// TwinCAT 3 PLC project PLC1
// Title: Example_project_GSBF
// Company: Gain Automation Technology B.V.
// Author: Gain Automation Technology
// ProjectVersion: 0.0.0.0
// Description: © 2025 Gain Automation Technology B.V. – MIT License
// ProgramVersion: 3.1.4026.19
// libraries:
//   GSBF_Common, * (Gain Automation Technology B.V.)
//   GSBF_HMI, * (Gain Automation Technology B.V.)
//   Tc2_Drive, * (Beckhoff Automation GmbH)
//   Tc2_EtherCAT, * (Beckhoff Automation GmbH)
//   Tc2_MC2, * (Beckhoff Automation GmbH)
//   Tc2_Standard, * (Beckhoff Automation GmbH)
//   Tc2_System, * (Beckhoff Automation GmbH)
//   Tc3_Module, * (Beckhoff Automation GmbH)
//   VisuDialogs, * (System)
//   VisuSymbols, 4.5.0.0 (System)
// project tree:
//   / GlobalTextList.TcGTLO, PlcTask.TcTTO, Visualization Manager.TcVMO (not stored)
//   GVLs/ GVL_Modules.TcGVL
//   POUs/1_Management_Layer/ ST_HmiAlarmList.TcDUT, FB_HMI_AlarmCollector.TcPOU
//   POUs/2_Units/UN_Machine/DUTs/ ST_UN_Machine_Hmi.TcDUT
//   POUs/2_Units/UN_Machine/ UN_Machine.TcPOU
//   POUs/3_Equipment_Modules/EM_InfeedConveyor/ EM_InfeedConveyor.TcPOU
//   POUs/3_Equipment_Modules/EM_InfeedConveyor/_DUTs/ E_EM_InfeedConveyor_Seq_ProductionExecute.TcDUT, E_EM_InfeedConveyor_Seq_ProductionStarting.TcDUT, ST_CommInfeedToLift.TcDUT, ST_CommLiftToInfeed.TcDUT, ST_EM_InfeedConveyor_Hmi.TcDUT
//   POUs/3_Equipment_Modules/EM_Lift/ EM_Lift.TcPOU
//   POUs/3_Equipment_Modules/EM_Lift/_DUTs/ E_EM_Lift_Seq_ProductionExecute.TcDUT, E_EM_Lift_Seq_StopServos.TcDUT, E_EM_Lift_Seq_ProductionStarting.TcDUT, ST_EM_Lift_Hmi.TcDUT
//   POUs/4_Control_Modules/CM_Door/ CM_Door.TcPOU
//   POUs/4_Control_Modules/CM_Door/_DUTs/ E_CM_Door_Seq_Logic.TcDUT, ST_CM_Door_Hmi.TcDUT
//   POUs/6_TwinCatChecks/ CheckBounds.TcPOU, CheckDivDInt.TcPOU, CheckDivLInt.TcPOU, CheckDivLReal.TcPOU, CheckDivReal.TcPOU, CheckLRangeSigned.TcPOU, CheckLRangeUnsigned.TcPOU, CheckPointer.TcPOU, CheckRangeSigned.TcPOU, CheckRangeUnsigned.TcPOU
//   POUs/ MAIN.TcPOU
//   VISUs/ HMI_Button.TcVIS, Header.TcVIS, Page_Main.TcVIS, Page_Alarms.TcVIS, Page_Infeed.TcVIS, Page_PackML.TcVIS, Visualization.TcVIS
// real-time tasks:
//   TASK PlcTask: cycle T#10ms, priority 20, ADS port 350
// motion (NC):
//   TASK NC-Task 1 SAF: cycle T#2ms, priority 4, ADS port 501
//   TASK NC-Task 1 SVB: cycle T#10ms, priority 8, ADS port 511
//   AXIS EM_Lift_Servo (id 1)
//     Dynamic: Jerk=22500
//     OtherSettings: AllowMotionCmdToSlave=true
//     encoder EncType=1
//     drive DrvType=5
//       Analog: TorqueSetpointScale=10, ScaleFactorActTorque=0.1
//       TimeComp: TaskDelayCycles=1
//     controller CtrType=1
//       CtrPara: PriorControlFactor=1
//         Observer: BandWidth=20
//   AXIS EM_LogicExample1_AxisVM (id 2)
//     Dynamic: Jerk=22500
//     OtherSettings: AllowMotionCmdToSlave=true
//     encoder EncType=1
//     drive DrvType=5
//       Analog: TorqueSetpointScale=10, ScaleFactorActTorque=0.1
//       TimeComp: TaskDelayCycles=1
//     controller CtrType=1
//       CtrPara: PriorControlFactor=1
//         Observer: BandWidth=20
//   AXIS EM_LogicExample2_Axis1 (id 4)
//     Dynamic: Jerk=22500
//     OtherSettings: AllowMotionCmdToSlave=true
//     encoder EncType=1
//     drive DrvType=5
//       Analog: TorqueSetpointScale=10, ScaleFactorActTorque=0.1
//       TimeComp: TaskDelayCycles=1
//     controller CtrType=1
//       CtrPara: PriorControlFactor=1
//         Observer: BandWidth=20
//   AXIS EM_LogicExample2_AxisVM (id 3)
//     Dynamic: Jerk=22500
//     OtherSettings: AllowMotionCmdToSlave=true
//     encoder EncType=1
//     drive DrvType=5
//       Analog: TorqueSetpointScale=10, ScaleFactorActTorque=0.1
//       TimeComp: TaskDelayCycles=1
//     controller CtrType=1
//       CtrPara: PriorControlFactor=1
//         Observer: BandWidth=20
// I/O:
//   DEVICE Device 1 (EtherCAT) (disabled), AmsNetId 169.254.247.113.2.1
//     Term 1 (EK1100) [EK1100 EtherCAT Coupler (2A E-Bus)]
//       Term 4 (EL1918) [EL1918, 8Ch. Safety Input 24V, TwinSAFE]
//         modules: Module 2 (FSLOGIC)
//       Term 3 (EL1904) [EL1904, 4 Ch. Safety Input 24V, TwinSAFE]
//         modules: Module 1 (FSOES)
//       Term 2 (EL2912) [EL2912, 2Ch. Safety Output 24V, 2A, TwinSAFE]
//         modules: Module 1 (FSOE), Module 2 (FSOUT), Module 3 (DEVICEIO), Module 4 (FSLOGIC)
// variable links:
//   (this object) <-> Device 1 (EtherCAT)/Term 1 (EK1100)/Term 3 (EL1904)
//     Term 1 (EK1100)/Term 4 (EL1918)/ConnectionInputs/Message_4 TxPDO <-> Module 1 (FSOES)/RxPDO/FSOE
//     Term 1 (EK1100)/Term 4 (EL1918)/ConnectionOutputs/Message_4 RxPDO <-> Module 1 (FSOES)/TxPDO/FSOE
//   (this object) <-> Device 1 (EtherCAT)/Term 1 (EK1100)/Term 4 (EL1918)
//     Term 1 (EK1100)/Term 3 (EL1904)/Module 1 (FSOES)/RxPDO/FSOE <-> ConnectionInputs/Message_4 TxPDO
//     Term 1 (EK1100)/Term 3 (EL1904)/Module 1 (FSOES)/TxPDO/FSOE <-> ConnectionOutputs/Message_4 RxPDO
//   PLC1 Instance <-> NC-Task 1 SAF/Axes/EM_Lift_Servo
//     PlcTask Inputs/GVL_Modules.g_emLift.s_cmMotorLift.IQ_Axis.NcToPlc <-> Outputs/ToPlc
//     PlcTask Outputs/GVL_Modules.g_emLift.s_cmMotorLift.IQ_Axis.PlcToNc <-> Inputs/FromPlc

CONFIGURATION PLC1
    RESOURCE PLC ON TwinCAT3
        TASK PlcTask(INTERVAL := T#10ms, PRIORITY := 20);
        PROGRAM MAIN WITH PlcTask : MAIN;
    END_RESOURCE
END_CONFIGURATION

// ---- POUs/1_Management_Layer/ST_HmiAlarmList.TcDUT
TYPE ST_HmiAlarmList :
STRUCT
	asAlarmList				: ARRAY[1..Param_Alarms.c_nMaxNrOfListEntries] OF STRING; // Active alarm texts for HMI list.
	sHighestActiveAlarm		: STRING; // Highest severity active alarm text.
END_STRUCT
END_TYPE

// ---- POUs/2_Units/UN_Machine/DUTs/ST_UN_Machine_Hmi.TcDUT
TYPE ST_UN_Machine_Hmi :
STRUCT
	// Local var
	fbHmiAlarmCollector		: FB_HMI_AlarmCollector;

END_STRUCT
END_TYPE

// ---- POUs/3_Equipment_Modules/EM_InfeedConveyor/_DUTs/E_EM_InfeedConveyor_Seq_ProductionExecute.TcDUT
{attribute 'qualified_only'}
{attribute 'strict'}
{attribute 'to_string'}
TYPE E_EM_InfeedConveyor_Seq_ProductionExecute :
(
	Idle := c_nSeqIdle, // Wait for production start or preconditions.
	Start := c_nSeqStart, // Select initial step based on sensors/door state.
	
	WaitForProduct, // Wait for product at start sensor.
	
	MoveProductToDoor, // Run belt to move product to end sensor.
	WaitUntilLiftReady, // Wait for lift at infeed position.
	RequestLiftReceiving, // Request lift to receive product.
	OpenDoor, // Open door before transfer.
	MoveProductInLift, // Run belt until lift confirms receipt.
	CloseDoor, // Close door after transfer.
	
	
	
	Ready := c_nSeqReady, // Sequence complete.
	Error := c_nSeqError // Sequence error handling.

);
END_TYPE

// ---- POUs/3_Equipment_Modules/EM_InfeedConveyor/_DUTs/E_EM_InfeedConveyor_Seq_ProductionStarting.TcDUT
{attribute 'qualified_only'}
{attribute 'strict'}
{attribute 'to_string'}
TYPE E_EM_InfeedConveyor_Seq_ProductionStarting :
(
	Idle := c_nSeqIdle, // Wait for PackML start command.
	Start := c_nSeqStart, // Decide open/close door at startup.
	
	OpenDoor, // Open door and wait for feedback.
	CloseDoor, // Close door and wait for feedback.
	
	Ready := c_nSeqReady, // Start sequence complete.
	Error := c_nSeqError // Start sequence error handling.

);
END_TYPE

// ---- POUs/3_Equipment_Modules/EM_InfeedConveyor/_DUTs/ST_CommInfeedToLift.TcDUT
TYPE ST_CommInfeedToLift :
STRUCT
	bReqExportProduct : BOOL; // Request lift to receive product from infeed.
	bBusyWithLift : BOOL; // Infeed busy with lift transfer (handshake/locking).
END_STRUCT
END_TYPE

// ---- POUs/3_Equipment_Modules/EM_InfeedConveyor/_DUTs/ST_CommLiftToInfeed.TcDUT
TYPE ST_CommLiftToInfeed :
STRUCT
	bAtInfeedPos : BOOL; // Lift is positioned at the infeed transfer point.
	bReadyForReceiving : BOOL; // Lift is ready to receive a product.
	bProductReceived : BOOL; // Lift confirms product has been received.
END_STRUCT
END_TYPE

// ---- POUs/3_Equipment_Modules/EM_InfeedConveyor/_DUTs/ST_EM_InfeedConveyor_Hmi.TcDUT
TYPE ST_EM_InfeedConveyor_Hmi :
STRUCT
	fbBelt : HMI_CM_MotorDol; // HMI controls for the infeed belt.
END_STRUCT
END_TYPE

// ---- POUs/3_Equipment_Modules/EM_Lift/_DUTs/E_EM_Lift_Seq_ProductionExecute.TcDUT
{attribute 'qualified_only'}
{attribute 'strict'}
{attribute 'to_string'}
TYPE E_EM_Lift_Seq_ProductionExecute :
(
	Idle := c_nSeqIdle, // Wait for production to start.
	Start := c_nSeqStart, // Begin production sequence steps.

	
	
	Ready := c_nSeqReady, // Sequence complete.
	Error := c_nSeqError // Sequence error handling.

);
END_TYPE

// ---- POUs/3_Equipment_Modules/EM_Lift/_DUTs/E_EM_Lift_Seq_StopServos.TcDUT
{attribute 'qualified_only'}
{attribute 'strict'}
{attribute 'to_string'}
TYPE E_EM_Lift_Seq_StopServos :
(
	Idle := c_nSeqIdle, // Wait for stop request.
	Start := c_nSeqStart, // Begin stop sequence (triggers EMR stop in logic).

	StopServo, // Reserved step for explicit stop if sequence is expanded.
	PowerOffServo, // Remove drive power after stop.
	
	
	Ready := c_nSeqReady, // Stop sequence complete.
	Error := c_nSeqError // Stop sequence error handling.

);
END_TYPE

// ---- POUs/3_Equipment_Modules/EM_Lift/_DUTs/E_EM_Lift_Seq_ProductionStarting.TcDUT
{attribute 'qualified_only'}
{attribute 'strict'}
{attribute 'to_string'}
TYPE E_EM_Lift_Seq_ProductionStarting :
(
	Idle := c_nSeqIdle, // Wait for PackML start command.
	Start := c_nSeqStart, // Decide whether to home or enable drive.
	
	
	ReferenceDrive, // Perform homing/reference procedure.
	EnableDrive, // Power on servo drive.
	MoveToStartPos, // Move to defined start position.
	
	Ready := c_nSeqReady, // Start sequence complete.
	Error := c_nSeqError // Start sequence error handling.

);
END_TYPE

// ---- POUs/3_Equipment_Modules/EM_Lift/_DUTs/ST_EM_Lift_Hmi.TcDUT
TYPE ST_EM_Lift_Hmi :
STRUCT
	fbMotorLift : HMI_CM_Servo; // HMI controls for the lift servo.
END_STRUCT
END_TYPE

// ---- POUs/4_Control_Modules/CM_Door/_DUTs/E_CM_Door_Seq_Logic.TcDUT
{attribute 'qualified_only'}
{attribute 'strict'}
{attribute 'to_string'}
TYPE E_CM_Door_Seq_Logic :
(
	Idle := c_nSeqIdle, // Wait for sequence start.
	Start := c_nSeqStart, // Decide operational vs disabled based on enable.
	
	Disabled, // Module disabled; wait for enable.
	Operational, // Normal door control logic active.
	
	Ready := c_nSeqReady, // Placeholder for ready state (unused in current logic).
	Error := c_nSeqError // Error state; stop motor and wait for clear.
);
END_TYPE

// ---- POUs/4_Control_Modules/CM_Door/_DUTs/ST_CM_Door_Hmi.TcDUT
TYPE ST_CM_Door_Hmi :
STRUCT
	btnCloseDoor : FB_HmiButton; // HMI button: request door close.
	btnOpenDoor : FB_HmiButton; // HMI button: request door open.
	btnStopDoor : FB_HmiButton; // HMI button: request door stop.
	bStaDoorOpen : BOOL; // Status: door open feedback.
	bStaDoorCLosed : BOOL; // Status: door closed feedback.
END_STRUCT
END_TYPE

// ---- GVLs/GVL_Modules.TcGVL
{attribute 'qualified_only'}
VAR_GLOBAL
	
// Management
	g_fbMachCtrlsManager	: FB_MachineControlsManager;
	g_fbHmiMachCtrlsManager	: FB_HMI_MachineControlsManager_StartStopMode;
	g_fbPackMLstatusManager	: FB_PackML_StatusManager;

	
// Units
	g_unMachine				: UN_Machine;
	
// Equipment modules
	g_emInfeedConveyor		: EM_InfeedConveyor;
	g_emLift 				: EM_Lift;
END_VAR

// ---- POUs/MAIN.TcPOU
PROGRAM MAIN 
VAR
END_VAR


// Main program cycle: call top-level managers and units in a clear order.
// Keep this list small; detailed behavior belongs inside the modules.

// PackML status manager
// Collects and aggregates PackML status for the system.
GVL_Modules.g_fbPackMLstatusManager();
	
// Machine controls manager
// HMI manager translates user actions into machine control requests.
GVL_Modules.g_fbHmiMachCtrlsManager(
	i_itfMachineControl := GVL_Modules.g_fbMachCtrlsManager); // Link HMI to machine controls.
// Machine controls manager coordinates PackML state requests for the unit.
GVL_Modules.g_fbMachCtrlsManager(
	i_itfModule := GVL_Modules.g_unMachine); // Link controls to the unit interface.
	
// Units
// Call each unit FB with system-level flags and managers.
GVL_Modules.g_unMachine(
	i_bReqEnable				:= TRUE, // Master enable for the unit (replace with safety chain if needed).
	i_bReqReset					:= GVL_Modules.g_fbMachCtrlsManager.p_bReset, // Reset request from machine controls.
	i_bReqSimulation			:= TRUE, // Simulation mode flag (toggle for real hardware).
	i_itfPackML_Parent			:= GVL_Modules.g_fbPackMLstatusManager, // PackML status manager.
	i_itfAlarmCollector_Parent	:= ); // Optional alarm manager interface.

END_PROGRAM

// ---- POUs/2_Units/UN_Machine/UN_Machine.TcPOU
FUNCTION_BLOCK UN_Machine EXTENDS FB_UN_PackML_Base
VAR_INPUT
END_VAR
VAR_OUTPUT
END_VAR
VAR
	// HMI
	s_stHmi : ST_UN_Machine_Hmi; // HMI structure (status and manual controls).
	
END_VAR

// Call Super
// Basemodule calls the following base method by calling SUPER^(): 
// - m_Main
// Add module-specific cyclic logic before/after SUPER^() if required.

SUPER^();

METHOD PROTECTED _m_Aborted : BOOL (* Return state complete when state is ready*)
VAR_INPUT
	(*First cycle of this state*)
	i_bCmdRestart	: BOOL;
	i_eActMode	: GSBF_Common.E_PackML_Mode;
END_VAR
// Allow clear when alarms are below critical.
// Add extra abort handling here if required.
IF s_fbAlarmCollector.p_eAlarmState < E_Alarm_Severity.Critical THEN
	s_fbPackML.m_ReqClear(); // Request clear of PackML state.
END_IF
END_METHOD

METHOD PROTECTED _m_Alarms
// Call base alarm handling.
SUPER^._m_Alarms();

// Add unit-level alarm conditions here if needed.
END_METHOD

METHOD PROTECTED _m_Hmi
// Call base HMI handling.
SUPER^._m_Hmi();

// Expose alarm collector to HMI for diagnostics.
s_stHmi.fbHmiAlarmCollector(i_itfAlarmCollector := s_fbAlarmCollector);
END_METHOD

METHOD PROTECTED _m_Logic
// Call base logic.
SUPER^._m_Logic();

// Unit-specific logic goes here (coordination between modules).
// Call HMI handling as part of the logic cycle.
_m_Hmi();
END_METHOD

METHOD PROTECTED _m_Modules
// Call base module handling.
SUPER^._m_Modules();

// Call infeed conveyor module and link to lift handshake.
GVL_Modules.g_emInfeedConveyor(
	i_bReqEnable					:= TRUE, // Enable module (replace with safety chain if needed).
	i_bReqReset						:= s_fbAlarmCollector.q_bReqReset, // Reset from alarm collector.
	i_bStaSafetyOk					:= TRUE, // Safety chain OK (replace with real input).
	i_bReqSimulation				:= p_bReqSimulation, // Simulation flag from unit.
	i_itfPackML_Parent				:= s_fbPackML, // PackML parent interface.
	i_itfAlarmCollector_Parent		:= s_fbAlarmCollector, // Alarm collector parent.
	q_stStaPackML					=> , // Optional PackML status feedback.
	i_stFromLift					:= GVL_Modules.g_emLift.q_stFromLift); // Lift status to infeed.

// Call lift module and link to infeed handshake.
GVL_Modules.g_emLift(
	i_bReqEnable:= TRUE, // Enable module (replace with safety chain if needed).
	i_bReqReset:= s_fbAlarmCollector.q_bReqReset, // Reset from alarm collector.
	i_bStaSafetyOk:= TRUE, // Safety chain OK (replace with real input).
	i_bReqSimulation:= p_bReqSimulation, // Simulation flag from unit.
	i_itfPackML_Parent:= s_fbPackML, // PackML parent interface.
	i_itfAlarmCollector_Parent:= s_fbAlarmCollector, // Alarm collector parent.
	q_stStaPackML=> , // Optional PackML status feedback.
	i_stToLift:= GVL_Modules.g_emInfeedConveyor.q_stToLift, // Infeed commands to lift.
	q_stFromLift=> ); // Lift status output.
END_METHOD

METHOD PROTECTED _m_Stopped : BOOL (* Return state complete when state is ready*)
VAR_INPUT
	(*First cycle of this state*)
	i_bCmdRestart	: BOOL;
	i_eActMode	: GSBF_Common.E_PackML_Mode;
END_VAR
// Allow reset when alarms are below error level.
// Add extra stopped-state logic here if required.
IF s_fbAlarmCollector.p_eAlarmState < E_Alarm_Severity.Error THEN
	s_fbPackML.m_ReqReset(); // Request PackML reset.
END_IF
END_METHOD

METHOD PUBLIC m_Main
// Main entry point for the unit.
// Use this to wrap additional high-level logic around base behavior.
SUPER^.m_Main();
END_METHOD

END_FUNCTION_BLOCK

// ---- POUs/3_Equipment_Modules/EM_InfeedConveyor/EM_InfeedConveyor.TcPOU
FUNCTION_BLOCK EM_InfeedConveyor EXTENDS FB_EM_PackML_Base
VAR_INPUT
	i_stFromLift : ST_CommLiftToInfeed; // Status/handshake from lift to infeed.
END_VAR
VAR_OUTPUT
	q_stToLift : ST_CommInfeedToLift; // Commands/handshake from infeed to lift.
END_VAR
VAR
	// Variables
	s_stHmi : ST_EM_InfeedConveyor_Hmi;	// HMI structure (status and manual controls).

	// Control modules
	s_cmBelt : CM_MotorDol; // Belt drive for infeed conveyor.
	s_cmHmiBelt : HMI_CM_MotorDol; // HMI helper for belt controls.
	
	s_cmDoor : CM_Door; // Door control module between conveyor and lift.
	
	
	// in/outputs
	s_diStartConveyor : FB_DigitalInput; // Sensor at conveyor start (product present).
	s_diEndConveyor : FB_DigitalInput; // Sensor at conveyor end (near lift).
	
	// Alarms
	s_fbAlmDoorOpenWithoutPermission : FB_AlarmHandler; // Door open while lift not at infeed.
	s_fbAlmUnexpectProductEndConveyor : FB_AlarmHandler; // Unexpected product detected at end sensor.
	
END_VAR

// Call Super
// Basemodule calls the following base method by calling SUPER^(): 
// - m_Main
// Add module-specific cyclic logic before/after SUPER^() if required.

SUPER^();

METHOD PROTECTED _m_Aborting : BOOL // Return state complete when state is ready
VAR_INPUT
	i_bCmdRestart	: BOOL;	//First cycle of this state
	i_eActMode 		: E_PackML_Mode;
END_VAR
// Stop door.
// Aborting should leave the module in a safe, passive state.
// Add any extra abort actions here (e.g., stop belt, clear outputs).
_m_Aborting	:= s_cmDoor.m_Stop();
END_METHOD

(* Collect alarm conditions from sub-modules. *)
METHOD PROTECTED _m_Alarms
(* All module alarms are handled in this method *)
(*==========================================================================================================*)
// Call base
SUPER^._m_Alarms();

// Add module-specific alarm conditions below.


// Door opened while lift is not at infeed position.
s_fbAlmDoorOpenWithoutPermission(
	i_bCmdRaise:= NOT i_stFromLift.bAtInfeedPos AND NOT s_cmDoor.p_bStaDoorClosed, 
	i_sMessage:= , 
	i_itfAlarmCollector:= p_itfAlarmCollector);

// Unexpected product detected at end sensor (raised explicitly elsewhere).
s_fbAlmUnexpectProductEndConveyor(
	i_bCmdRaise:= , // leave empty, this alarm is set by m_Raise 
	i_sMessage:= , 
	i_itfAlarmCollector:= p_itfAlarmCollector);
END_METHOD

METHOD PROTECTED _m_Execute : BOOL // Return state complete when state is ready
VAR_INPUT
	i_bCmdRestart	: BOOL;	//First cycle of this state
	i_eActMode 		: E_PackML_Mode;
END_VAR
// Execute production sequence only in Production mode.
// For other modes, return TRUE or add mode-specific behavior.
IF i_eActMode = E_PackML_Mode.Production THEN
	_m_Execute := _m_ProductionExecute(i_bCmdRestart := i_bCmdRestart).p_bStaReady;
ELSE
	_m_Execute := TRUE;
END_IF
END_METHOD

METHOD PROTECTED _m_Hmi
// Expose belt controls to the HMI in Manual mode.
// Extend this method with extra HMI controls or status fields as needed.
s_stHmi.fbBelt(
	i_bReqEnableHmiControls:= s_fbPackML.p_eActMode = E_PackML_Mode.Manual, // Enable manual HMI buttons in Manual mode.
	i_itfCM_MotorDol:= s_cmBelt);
END_METHOD

(* Initialization, set initial data. *)
METHOD PROTECTED _m_Init
// Call base
SUPER^._m_Init();

// Configure alarms and initial module parameters here.
// Alarms
s_fbAlmDoorOpenWithoutPermission.p_itfConfig.p_bCfgAutoReset		:= FALSE;                                                
s_fbAlmDoorOpenWithoutPermission.p_itfConfig.p_bCfgEnable			:= TRUE;                                                   
s_fbAlmDoorOpenWithoutPermission.p_itfConfig.p_eCfgSeverity			:= E_Alarm_Severity.Error;                             
s_fbAlmDoorOpenWithoutPermission.p_itfConfig.p_tmCfgDelay			:= T#0S;                                                   
s_fbAlmDoorOpenWithoutPermission.p_itfConfig.p_stCfgEventEntry		:= TC_EVENTs.EM_InfeedConveyor_EventClass.AlmDoorOpenWithoutPermission;

s_fbAlmUnexpectProductEndConveyor.p_itfConfig.p_bCfgAutoReset		:= FALSE;                                                
s_fbAlmUnexpectProductEndConveyor.p_itfConfig.p_bCfgEnable			:= TRUE;                                                   
s_fbAlmUnexpectProductEndConveyor.p_itfConfig.p_eCfgSeverity		:= E_Alarm_Severity.Error;                             
s_fbAlmUnexpectProductEndConveyor.p_itfConfig.p_tmCfgDelay			:= T#0S;                                                   
s_fbAlmUnexpectProductEndConveyor.p_itfConfig.p_stCfgEventEntry		:= TC_EVENTs.EM_InfeedConveyor_EventClass.AlmUnexpectProductEndConveyor;
END_METHOD

(* Process unit inputs. *)
METHOD PROTECTED _m_Inputs
// Call base 
SUPER^._m_Inputs();

// Map IO or communication inputs to internal status here.
// Call inputs
s_diStartConveyor(); // Start sensor at infeed side.
s_diEndConveyor(); // End sensor at lift side.
END_METHOD

(* Call sub-modules (equipment and/or control modules). *)
METHOD PROTECTED _m_Modules
// Call base
SUPER^._m_Modules();

// Call belt motor control module.
s_cmBelt(
	i_bReqEnable:= p_bReqEnable, 
	i_bReqReset:= , // Add extra reset command, normally reset is done by alarmcollector. 
	i_bReqSimulation:= p_bReqSimulation, 
	i_itfAlarmCollector_Parent:= p_itfAlarmCollector); // Propagate belt alarms to module.
	
// Call door control module and pass common flags.
s_cmDoor(
	i_bReqEnable:= p_bReqEnable, 
	i_bReqReset:= , // Add extra reset command, normally reset is done by alarmcollector.
	i_bReqEnableHmiControls:= s_fbPackML.p_eActMode = E_PackML_Mode.Manual, 
	i_bReqSimulation:= p_bReqSimulation, 
	i_itfAlarmCollector_Parent:= p_itfAlarmCollector); // Propagate door alarms to module.
END_METHOD

METHOD _m_ProductionExecute : ITF_FB_SeqControl
VAR_INPUT
	i_bCmdRestart : BOOL;
END_VAR
VAR_INST
	s_fbSeqControl  : FB_SeqControl;
	s_eSeq 			: E_EM_InfeedConveyor_Seq_ProductionExecute;
END_VAR
// Sequencer bookkeeping (current step and entry handling).
s_fbSeqControl(
	i_bReqStart:= i_bCmdRestart, // Start sequencer on first cycle of state.
	i_rnActSeqStep:= s_eSeq, // Active step enum.
	i_sActSeqStep:= TO_STRING(s_eSeq)); // Step name for logging/trace.


// Production sequencer - implement the automatic infeed flow here.
CASE s_eSeq OF
	E_EM_InfeedConveyor_Seq_ProductionExecute.Idle:
		// Wait for production to start or for preconditions.
		// Clear transient outputs here if required (requests, flags).
		;
		
	E_EM_InfeedConveyor_Seq_ProductionExecute.Start:
		// Choose initial step based on current conveyor/door state.
		// This avoids moving product or door unnecessarily at startup.
		IF s_cmDoor.p_bStaDoorClosed AND s_diEndConveyor.p_bStaValue THEN
			// Product already at end and door closed: wait for lift.
			s_fbSeqControl.m_ReqStep(E_EM_InfeedConveyor_Seq_ProductionExecute.WaitUntilLiftReady); // Product at end, wait for lift.
		ELSIF s_cmDoor.p_bStaDoorOpen THEN
			// Door open: request lift to receive immediately.
			s_fbSeqControl.m_ReqStep(E_EM_InfeedConveyor_Seq_ProductionExecute.RequestLiftReceiving);	// Door open, request lift now.
		ELSE
			// Default: wait for product at start sensor.
			s_fbSeqControl.m_ReqStep(E_EM_InfeedConveyor_Seq_ProductionExecute.WaitForProduct);	// Default: wait for product.
		END_IF		
	
	E_EM_InfeedConveyor_Seq_ProductionExecute.WaitForProduct:
		// Wait until a product arrives at the start sensor.
		// Add debouncing or filtering here if required by the hardware.
		IF s_diStartConveyor.p_bStaValue THEN
			s_fbSeqControl.m_ReqStep(E_EM_InfeedConveyor_Seq_ProductionExecute.MoveProductToDoor); // Product detected at start.
		ELSIF s_diEndConveyor.p_bStaValue THEN
			// Product detected at end without running belt -> unexpected.
			s_fbAlmUnexpectProductEndConveyor.m_CmdRaise(); // Raise alarm for unexpected product.
			
			// No transition; PackML will handle the alarm state.
		END_IF
	
	E_EM_InfeedConveyor_Seq_ProductionExecute.MoveProductToDoor:
		// Move product towards the door until end sensor is active.
		// Add jam detection or timeout here if the belt should not run too long.
		IF NOT s_diEndConveyor.p_bStaValue THEN
			// Run belt until product is at end of conveyor.
			s_cmBelt.m_StartFwd(); // Run belt forward.
		ELSE
			// Product is at end conveyor, stop belt.
			IF s_cmBelt.m_Stop() THEN // Stop belt before requesting lift.
				s_fbSeqControl.m_ReqStep(E_EM_InfeedConveyor_Seq_ProductionExecute.WaitUntilLiftReady);
			END_IF
		END_IF
	
	E_EM_InfeedConveyor_Seq_ProductionExecute.WaitUntilLiftReady:
		// Wait until lift is positioned at infeed.
		// Add timeout and alarm handling here if required.
		IF i_stFromLift.bAtInfeedPos THEN
			s_fbSeqControl.m_ReqStep(E_EM_InfeedConveyor_Seq_ProductionExecute.RequestLiftReceiving); // Lift in position.
		END_IF	
			 
	E_EM_InfeedConveyor_Seq_ProductionExecute.RequestLiftReceiving:
		// Handshake: request lift to receive product.
		q_stToLift.bReqExportProduct := TRUE; // Request lift to receive product.
		// Keep this request TRUE while in this step; clear it in other steps if needed.
		
		// Continue once lift confirms it is ready.
		IF i_stFromLift.bReadyForReceiving THEN
			s_fbSeqControl.m_ReqStep(E_EM_InfeedConveyor_Seq_ProductionExecute.OpenDoor); // Lift ready.
		END_IF
		
	E_EM_InfeedConveyor_Seq_ProductionExecute.OpenDoor:
		// Open door before transferring product into lift.
		// Add interlocks here if the door should not open in certain conditions.
		IF s_cmDoor.m_OpenDoor() THEN // Command door open and wait for feedback.
			s_fbSeqControl.m_ReqStep(E_EM_InfeedConveyor_Seq_ProductionExecute.MoveProductInLift);
		END_IF
		
	E_EM_InfeedConveyor_Seq_ProductionExecute.MoveProductInLift:
		// Drive belt until lift reports product received.
		// Add timeout or sensor validation to detect mis-transfer.
		IF NOT i_stFromLift.bProductReceived THEN // Keep feeding until lift confirms receipt.
			// Belt on.
			s_cmBelt.m_StartFwd(); // Move product into lift.
		ELSE	
			// Product in lift, stop conveyor.
			s_cmBelt.m_Stop(); // Stop belt once received.
			
			s_fbSeqControl.m_ReqStep(E_EM_InfeedConveyor_Seq_ProductionExecute.CloseDoor); // Secure door after transfer.
		END_IF
		
	E_EM_InfeedConveyor_Seq_ProductionExecute.CloseDoor:
		// Close door and return to waiting for next product.
		// Add checks for door blocked or safety conditions if required.
		IF s_cmDoor.m_CloseDoor() THEN // Command door close and wait for feedback.
			s_fbSeqControl.m_ReqStep(E_EM_InfeedConveyor_Seq_ProductionExecute.WaitForProduct); // Ready for next product.
		END_IF
		
	E_EM_InfeedConveyor_Seq_ProductionExecute.Ready:
		// Sequence complete; keep outputs stable.
		;
	E_EM_InfeedConveyor_Seq_ProductionExecute.Error:
		// Handle recoverable errors or trigger alarms here.
		;
END_CASE

// Return sequencer status to PackML state handler.
_m_ProductionExecute := s_fbSeqControl.m_getResult(TO_STRING(s_eSeq)); // Return sequencer status.
END_METHOD

METHOD _m_ProductionStarting : ITF_FB_SeqControl
VAR_INPUT
	i_bCmdRestart : BOOL;
END_VAR
VAR_INST
	s_fbSeqControl  : FB_SeqControl;
	s_eSeq 			: E_EM_InfeedConveyor_Seq_ProductionStarting;
END_VAR

// Sequencer bookkeeping (current step and entry handling).
s_fbSeqControl(
	i_bReqStart:= i_bCmdRestart, // Start sequencer on first cycle of state.
	i_rnActSeqStep:= s_eSeq, // Active step enum.
	i_sActSeqStep:= TO_STRING(s_eSeq)); // Step name for logging/trace.
	
// Production start sequence: set door to a known safe state.
CASE s_eSeq OF 
	E_EM_InfeedConveyor_Seq_ProductionStarting.Idle:
		// Wait for start command from PackML.
		// Clear transient outputs here if required (requests, flags).
		;
	E_EM_InfeedConveyor_Seq_ProductionStarting.Start:
		// Decide whether door should be opened or closed at startup.
		// Replace with actual "product present" logic if available.
		IF s_cmDoor.p_bStaDoorBlocked THEN
			s_fbSeqControl.m_ReqStep(E_EM_InfeedConveyor_Seq_ProductionStarting.OpenDoor); // Door blocked, open at start.
		ELSE 
			s_fbSeqControl.m_ReqStep(E_EM_InfeedConveyor_Seq_ProductionStarting.CloseDoor); // Otherwise close at start.
		END_IF
		
		
	E_EM_InfeedConveyor_Seq_ProductionStarting.OpenDoor:
		// Open door at startup (e.g., product present at door).
		// Add interlocks or safety checks here if required.
		IF s_cmDoor.m_OpenDoor() THEN // Command door open and wait for feedback.
			s_fbSeqControl.m_ReqStep(E_EM_InfeedConveyor_Seq_ProductionStarting.Ready); // Startup complete.
		END_IF
	E_EM_InfeedConveyor_Seq_ProductionStarting.CloseDoor:

		// Close door at startup (e.g., no product present).
		// Add interlocks or safety checks here if required.
		IF s_cmDoor.m_CloseDoor() THEN // Command door close and wait for feedback.
			s_fbSeqControl.m_ReqStep(E_EM_InfeedConveyor_Seq_ProductionStarting.Ready); // Startup complete.
		END_IF
		
	E_EM_InfeedConveyor_Seq_ProductionStarting.Ready:
		// Start sequence complete; ready for Execute state.
		;
	E_EM_InfeedConveyor_Seq_ProductionStarting.Error:
		// Handle startup errors or request operator intervention here.
		;
END_CASE

// Return sequencer status to PackML state handler.
_m_ProductionStarting := s_fbSeqControl.m_getResult(TO_STRING(s_eSeq)); // Return sequencer status.
END_METHOD

METHOD PROTECTED _m_Starting : BOOL // Return state complete when state is ready
VAR_INPUT
	i_bCmdRestart	: BOOL;	//First cycle of this state
	i_eActMode 		: E_PackML_Mode;
END_VAR
VAR_INST
	s_fbSeqControl 	: FB_SeqControl;
	s_eSeq			: E_EM_InfeedConveyor_Seq_ProductionStarting;
END_VAR
// PackML Starting: run production-start sequencer in Production mode.
IF i_eActMode = E_PackML_Mode.Production THEN
	_m_Starting := _m_ProductionStarting(i_bCmdRestart := i_bCmdRestart).p_bStaReady;
ELSE
	_m_Starting := TRUE;
END_IF
END_METHOD

METHOD PROTECTED _m_Stopping : BOOL // Return state complete when state is ready
VAR_INPUT
	i_bCmdRestart	: BOOL;	//First cycle of this state
	i_eActMode 		: E_PackML_Mode;
END_VAR
// Stop door.
// Add belt stop or other safe-state actions if required.
_m_Stopping	:= s_cmDoor.m_Stop();
END_METHOD

END_FUNCTION_BLOCK

// ---- POUs/4_Control_Modules/CM_Door/CM_Door.TcPOU
FUNCTION_BLOCK CM_Door EXTENDS FB_CM_Base
VAR_INPUT
	i_bReqEnableHmiControls : BOOL;	// Request to enable HMI control buttons (open/close/stop).
END_VAR
VAR_OUTPUT
END_VAR
VAR
	// Control modules
	s_cmMotor : CM_MotorDol; // Door motor (forward=open, reverse=close).
 
	
	// in/outputs
	s_diDoorIsOpen : FB_DigitalInput; // Feedback: door open position.
	s_diDoorIsClosed : FB_DigitalInput; // Feedback: door closed position.
	s_diDoorIsBlocked : FB_DigitalInput; // Feedback: door blocked sensor.
	
	// Alarms
	
	s_fbAlmDoorIsBlocked : FB_AlarmHandler; // Blocked while moving.
	s_fbAlmFeedbackBothOn : FB_AlarmHandler; // Both open and closed feedback active.
	s_fbAlmDoorNotOpen : FB_AlarmHandler; // Door did not reach open position.
	s_fbAlmDoorNotClosed : FB_AlarmHandler;	// Door did not reach closed position.

	// Hmi
	s_stHmi : ST_CM_Door_Hmi; // HMI structure (buttons + status).
END_VAR

// Call base 
SUPER^();

(* Monitor alarm conditions. *)
METHOD PROTECTED _m_Alarms

SUPER^._m_Alarms();

// Feedback conflict: open and closed at the same time.
s_fbAlmFeedbackBothOn(
	i_bCmdRaise:= s_diDoorIsOpen.p_bStaValue AND s_diDoorIsClosed.p_bStaValue, 
	i_sMessage:= , 
	i_itfAlarmCollector:= p_itfAlarmCollector);
	
// Door blocked while motor runs.
s_fbAlmDoorIsBlocked(
	i_bCmdRaise:= NOT s_cmMotor.p_bStaStandstill AND s_diDoorIsBlocked.p_bStaValue, 
	i_sMessage:= , 
	i_itfAlarmCollector:= p_itfAlarmCollector);
	
// Door should open within delay when running forward.
s_fbAlmDoorNotOpen.p_itfConfig.p_tmCfgDelay := T#6S;	
s_fbAlmDoorNotOpen(
	i_bCmdRaise:= s_cmMotor.p_bStaRunningFwd AND NOT s_diDoorIsOpen.p_bStaValue, 
	i_sMessage:= , 
	i_itfAlarmCollector:= p_itfAlarmCollector);
	

// Door should close within delay when running reverse.
s_fbAlmDoorNotClosed.p_itfConfig.p_tmCfgDelay := T#6S;		
s_fbAlmDoorNotClosed(
	i_bCmdRaise:= s_cmMotor.p_bStaRunningRev AND NOT s_diDoorIsClosed.p_bStaValue, 
	i_sMessage:= , 
	i_itfAlarmCollector:= p_itfAlarmCollector);
END_METHOD

METHOD PROTECTED _m_Hmi
VAR_INPUT
END_VAR
VAR_INST
	s_bStaOpening : BOOL;
	s_bStaClosing : BOOL;
END_VAR



// Update HMI buttons with current enable/state.
s_stHmi.btnOpenDoor(
	i_bEnable:= i_bReqEnableHmiControls, 
	i_bProcessState:= s_bStaOpening);
	
s_stHmi.btnCloseDoor(
	i_bEnable:= i_bReqEnableHmiControls, 
	i_bProcessState:= s_bStaClosing);

s_stHmi.btnStopDoor(
	i_bEnable:= i_bReqEnableHmiControls);	
	
// Latch requested direction on rising edge.
IF s_stHmi.btnOpenDoor.q_bStateOsr THEN
	s_bStaOpening := TRUE;
	s_bStaClosing := FALSE;
END_IF	

IF s_stHmi.btnCloseDoor.q_bStateOsr THEN
	s_bStaOpening := FALSE;
	s_bStaClosing := TRUE;
END_IF	

// Stop request or error cancels movement.
IF s_stHmi.btnStopDoor.q_bStateOsr OR p_eAlarmState >= E_Alarm_Severity.Error THEN
	s_bStaOpening := FALSE;
	s_bStaClosing := FALSE;
	m_Stop();
END_IF	

// Execute open/close request until feedback is reached.
IF s_bStaOpening THEN
	IF m_OpenDoor() THEN
		s_bStaOpening := FALSE;
	END_IF
END_IF


IF s_bStaClosing THEN
	IF m_CloseDoor() THEN
		s_bStaClosing := FALSE;
	END_IF
END_IF

// Publish status to HMI.
s_stHmi.bStaDoorOpen := p_bStaDoorOpen;
s_stHmi.bStaDoorCLosed := p_bStaDoorClosed;
END_METHOD

(* Initialization, set initial data. *)
METHOD PROTECTED _m_Init
// Call base
SUPER^._m_Init();

// Alarms
s_fbAlmDoorIsBlocked.p_itfConfig.p_bCfgAutoReset		:= FALSE;                                                
s_fbAlmDoorIsBlocked.p_itfConfig.p_bCfgEnable			:= TRUE;                                                   
s_fbAlmDoorIsBlocked.p_itfConfig.p_eCfgSeverity			:= E_Alarm_Severity.Error;                             
s_fbAlmDoorIsBlocked.p_itfConfig.p_tmCfgDelay			:= T#0S;                                                   
s_fbAlmDoorIsBlocked.p_itfConfig.p_stCfgEventEntry		:= TC_EVENTS.Alarmen.CM_Door_AlmDoorIsBlocked;

s_fbAlmFeedbackBothOn.p_itfConfig.p_bCfgAutoReset		:= FALSE;                                                
s_fbAlmFeedbackBothOn.p_itfConfig.p_bCfgEnable			:= TRUE;                                                   
s_fbAlmFeedbackBothOn.p_itfConfig.p_eCfgSeverity			:= E_Alarm_Severity.Error;                             
s_fbAlmFeedbackBothOn.p_itfConfig.p_tmCfgDelay			:= T#0S;                                                   
s_fbAlmFeedbackBothOn.p_itfConfig.p_stCfgEventEntry		:= TC_EVENTS.Alarmen.CM_Door_AlmFeedbackBothOn;

s_fbAlmDoorNotOpen.p_itfConfig.p_bCfgAutoReset			:= FALSE;                                                
s_fbAlmDoorNotOpen.p_itfConfig.p_bCfgEnable				:= TRUE;                                                   
s_fbAlmDoorNotOpen.p_itfConfig.p_eCfgSeverity			:= E_Alarm_Severity.Error;                             
s_fbAlmDoorNotOpen.p_itfConfig.p_tmCfgDelay				:= T#0S;                                                   
s_fbAlmDoorNotOpen.p_itfConfig.p_stCfgEventEntry		:= TC_EVENTs.Alarmen.CM_Door_AlmDoorIsBlocked;

s_fbAlmDoorNotClosed.p_itfConfig.p_bCfgAutoReset		:= FALSE;                                                
s_fbAlmDoorNotClosed.p_itfConfig.p_bCfgEnable			:= TRUE;                                                   
s_fbAlmDoorNotClosed.p_itfConfig.p_eCfgSeverity			:= E_Alarm_Severity.Error;                             
s_fbAlmDoorNotClosed.p_itfConfig.p_tmCfgDelay			:= T#0S;                                                   
s_fbAlmDoorNotClosed.p_itfConfig.p_stCfgEventEntry		:= TC_EVENTs.Alarmen.CM_Door_AlmFeedbackBothOn;
END_METHOD

(* Read hardware and module inputs. If applicable, apply filtering, scaling and/or conversion to local variables. *) 
METHOD PROTECTED _m_Inputs
// Call base
SUPER^._m_Inputs();


// Call inputs
s_diDoorIsOpen();
s_diDoorIsClosed();
s_diDoorIsBlocked();
END_METHOD

(* Handle the internal logic of the control module. *)
METHOD PROTECTED _m_Logic
VAR_INST
	s_fbSeqControl : FB_SeqControl;
	s_eSeq : E_CM_Door_Seq_Logic;
END_VAR
// Call base
SUPER^._m_Logic();

_m_Hmi();

// Call modules
_m_Modules();

// Sequencer tracks the door state machine.
// Call sequencer
s_fbSeqControl(
	i_bReqStart:= FALSE, 
	i_rnActSeqStep:= s_eSeq, 
	i_sActSeqStep:= TO_STRING(s_eSeq));

// Logic
CASE s_eSeq OF 
	E_CM_Door_Seq_Logic.Idle:
		// Go to operational state
		s_fbSeqControl.m_ReqStep(E_CM_Door_Seq_Logic.Start);
		
	E_CM_Door_Seq_Logic.Start:

		IF NOT p_bReqEnable THEN
			// Disabled request takes priority.
			s_fbSeqControl.m_ReqStep(E_CM_Door_Seq_Logic.Disabled);
		ELSE
			// Start successful: go operational.
			s_fbSeqControl.m_ReqStep(E_CM_Door_Seq_Logic.Operational);
		END_IF
	
	E_CM_Door_Seq_Logic.Disabled:
		IF p_bReqEnable THEN
			// Re-enable sequence.
			s_fbSeqControl.m_ReqStep(E_CM_Door_Seq_Logic.Start);
		END_IF
	
		
	E_CM_Door_Seq_Logic.Operational:
		// Stop motor when door is open
		IF s_diDoorIsOpen.p_bStaValue 
			AND s_cmMotor.p_bStaRunningFwd 
		THEN
			m_Stop();
		END_IF
		
		// Stop motor when door is closed
		IF s_diDoorIsClosed.p_bStaValue 
			AND s_cmMotor.p_bStaRunningRev 
		THEN
			m_Stop();
		END_IF
		
	
	
		// Transition
		IF NOT p_bReqEnable THEN
			// Disabled request wins.
			s_fbSeqControl.m_ReqStep(E_CM_Door_Seq_Logic.Disabled);
		ELSIF p_eAlarmState >= E_Alarm_Severity.Error THEN
			// Some error is active, go to error state
			s_fbSeqControl.m_ReqStep(E_CM_Door_Seq_Logic.Error);
		END_IF


	
	E_CM_Door_Seq_Logic.Ready:
		;
		
	E_CM_Door_Seq_Logic.Error:
		// Stop motor
		m_Stop();
	
		// Transition 
		IF NOT p_bReqEnable THEN
			s_fbSeqControl.m_ReqStep(E_CM_Door_Seq_Logic.Disabled);
		ELSIF p_eAlarmState < E_Alarm_Severity.Error THEN
			// Error cleared: restart sequence.
			s_fbSeqControl.m_ReqStep(E_CM_Door_Seq_Logic.Start);
		END_IF

END_CASE

s_fbSeqControl.m_Update(i_sActSeqStep := TO_STRING(s_eSeq));
END_METHOD

METHOD _m_Modules : BOOL
VAR_INPUT
END_VAR
// Call motor control module and connect to alarm collector.
s_cmMotor(
	i_bReqEnable:= p_bReqEnable, 
	i_bReqReset:= , // Can be leaved empty, is automatically done by alarmcollector
	i_bReqSimulation:= i_bReqSimulation, 
	i_itfAlarmCollector_Parent:= p_itfAlarmCollector);
END_METHOD

METHOD PROTECTED _m_Simulation
VAR_INST
	s_bSimDoorIsClosed : BOOL;
	s_bSimDoorIsOpen : BOOL;
	
	s_tonSimOpening : TON;
	s_tonSimClosing : TON;
END_VAR


// Simulate feedback timing based on motor direction.
s_tonSimOpening(in := s_cmMotor.p_bStaRunningFwd, PT := T#1MS);
s_tonSimClosing(in := s_cmMotor.p_bStaRunningRev, PT := T#5MS);

// When motor is running for x seconds set simulation status to open. 
IF s_tonSimOpening.Q THEN
	s_bSimDoorIsOpen := TRUE;
ELSIF s_cmMotor.p_bStaRunningRev THEN
	s_bSimDoorIsOpen := FALSE;	
END_IF

// When motor is running reverse long enough set simulation status to closed.
IF s_tonSimClosing.Q THEN
	s_bSimDoorIsClosed := TRUE;
ELSIF s_cmMotor.p_bStaRunningFwd THEN
	s_bSimDoorIsClosed := FALSE;	
END_IF

// Copy simulation value to IO
s_diDoorIsOpen.m_Simulation(i_bSimulate := p_bReqSimulation, i_bvalue := s_bSimDoorIsOpen);
s_diDoorIsClosed.m_Simulation(i_bSimulate := p_bReqSimulation, i_bvalue := s_bSimDoorIsClosed);
END_METHOD

METHOD m_CloseDoor : BOOL
VAR_INPUT
END_VAR
// Run reverse until closed feedback is active.
IF p_bReqEnable 
	AND p_eAlarmState < E_Alarm_Severity.Error 
	AND NOT s_diDoorIsClosed.p_bStaValue 
THEN
	// Start motor reverse
	s_cmMotor.m_StartRev();
ELSE
	s_cmMotor.m_Stop();
END_IF

m_CloseDoor := s_diDoorIsClosed.p_bStaValue;
END_METHOD

METHOD m_OpenDoor : BOOL
VAR_INPUT
END_VAR
// Run forward until open feedback is active.
IF p_bReqEnable 
	AND p_eAlarmState < E_Alarm_Severity.Error 
	AND NOT s_diDoorIsOpen.p_bStaValue 
THEN
	// Start motor forward
	s_cmMotor.m_StartFwd();
ELSE
	s_cmMotor.m_Stop();
END_IF

m_OpenDoor := s_diDoorIsOpen.p_bStaValue;
END_METHOD

METHOD m_Stop : BOOL
VAR_INPUT
END_VAR
// Stop motor and report standstill.
s_cmMotor.m_Stop();

m_Stop := s_cmMotor.p_bStaStandstill;
END_METHOD

PROPERTY p_bStaDoorBlocked : BOOL
GET
p_bStaDoorBlocked := s_diDoorIsBlocked.p_bStaValue;
END_GET
END_PROPERTY

PROPERTY PUBLIC p_bStaDoorClosed : BOOL
GET
p_bStaDoorClosed := s_diDoorIsClosed.p_bStaValue;
END_GET
END_PROPERTY

PROPERTY PUBLIC p_bStaDoorOpen : BOOL
GET
p_bStaDoorOpen := s_diDoorIsOpen.p_bStaValue;
END_GET
END_PROPERTY

END_FUNCTION_BLOCK

// ---- POUs/3_Equipment_Modules/EM_Lift/EM_Lift.TcPOU
FUNCTION_BLOCK EM_Lift EXTENDS FB_EM_PackML_Base
VAR_INPUT
	i_stToLift : ST_CommInfeedToLift; // Command from infeed to lift.
END_VAR
VAR_OUTPUT
	q_stFromLift : ST_CommLiftToInfeed; // Status from lift to infeed.
END_VAR
VAR
	// Variables
	s_stHmi : ST_EM_Lift_Hmi;	// HMI status and controls.


	// Control modules
	s_cmMotorLift : CM_ServoAX8000;	// Lift servo axis control.
	
END_VAR

// Call Super
// Basemodule calls the following base method by calling SUPER^(): 
// - m_Main
// Add module-specific cyclic logic before/after SUPER^() if required.

SUPER^();

METHOD PROTECTED _m_Aborting : BOOL // Return state complete when state is ready
VAR_INPUT
	i_bCmdRestart	: BOOL;	//First cycle of this state
	i_eActMode 		: E_PackML_Mode;
END_VAR
// Abort and disable servo
// Use stop-sequence to bring the lift axis to a safe state.
// Add any extra abort actions here (e.g., vent valves, set outputs).
_m_Aborting	:= _m_SeqStopServos(i_bCmdRestart := i_bCmdRestart).p_bStaReady;
END_METHOD

(* Collect alarm conditions from sub-modules. *)
METHOD PROTECTED _m_Alarms
(* All module alarms are handled in this method *)
(*==========================================================================================================*)
// Call base
SUPER^._m_Alarms();

// Add module-specific alarm conditions here and link them to the alarm collector.
END_METHOD

METHOD PROTECTED _m_Execute : BOOL // Return state complete when state is ready
VAR_INPUT
	i_bCmdRestart	: BOOL;	//First cycle of this state
	i_eActMode 		: E_PackML_Mode;
END_VAR
// Execute production sequence only in Production mode.
// For other modes, return TRUE or add mode-specific logic.
IF i_eActMode = E_PackML_Mode.Production THEN
	_m_Execute := _m_ProductionExecute(i_bCmdRestart := i_bCmdRestart).p_bStaReady;
ELSE
	_m_Execute := TRUE;
END_IF
END_METHOD

METHOD PROTECTED _m_Hmi
// Expose lift servo controls to the HMI in Manual mode.
// Extend this method with extra HMI widgets or status fields as needed.
s_stHmi.fbMotorLift(
	i_bReqEnableHmiControls:= s_fbPackML.p_eActMode = E_PackML_Mode.Manual, 
	i_itfCM_Servo:= s_cmMotorLift,
	i_eCfgMoveAbs:= E_HMI_CM_SERVO_MoveAbsMode_Direction.MoveToModuloPosShortestWay);
END_METHOD

(* Initialization, set initial data. *)
METHOD PROTECTED _m_Init
// Call base
SUPER^._m_Init();

// Initialize module-specific parameters and defaults here.
END_METHOD

(* Process unit inputs. *)
METHOD PROTECTED _m_Inputs
// Call base 
SUPER^._m_Inputs();

// Map IO or communication inputs to internal variables here.
END_METHOD

(* Call sub-modules (equipment and/or control modules). *)
METHOD PROTECTED _m_Modules
// Call base
SUPER^._m_Modules();

// Call lift servo control module and pass common flags.
// Adjust override, interlocks, and safety conditions to your machine.
s_cmMotorLift(
	i_bReqEnable:= p_bReqEnable, // Enable/reset/simulation are typically controlled by PackML/base module.
	i_bReqReset:= ,				 // done by alarmcollector 
	i_bReqSimulation:= p_bReqSimulation, 	// Connect alarm collector so servo alarms propagate to the module.
	i_itfAlarmCollector_Parent:= s_fbAlarmCollector, 
	i_bEmrStopOk:= TRUE, // Safety chain OK (replace with real E-Stop OK signal if available)
	i_fOverride:= 100, // Motion override in percent (100 = full speed).
	i_bDisableForward:= FALSE, // Direction/axis interlocks (set TRUE to block motion).
	i_bDisableReverse:= FALSE, // Direction/axis interlocks (set TRUE to block motion).
	i_bDisableAxis:= FALSE, 
	i_bExtReferenceSignal:= );	// Optional external reference signal (leave empty if unused).
END_METHOD

METHOD _m_ProductionExecute : ITF_FB_SeqControl
VAR_INPUT
	i_bCmdRestart : BOOL;
END_VAR
VAR_INST
	s_fbSeqControl  : FB_SeqControl;
	s_eSeq 			: E_EM_Lift_Seq_ProductionExecute;
END_VAR
// Sequencer bookkeeping (current step and entry handling).
s_fbSeqControl(
	i_bReqStart:= i_bCmdRestart, 
	i_rnActSeqStep:= s_eSeq, 
	i_sActSeqStep:= TO_STRING(s_eSeq));


// Production sequencer - implement the automatic process here.
CASE s_eSeq OF
	E_EM_Lift_Seq_ProductionExecute.Idle:
		// Wait for start conditions or upstream handshake.
		;
		
	E_EM_Lift_Seq_ProductionExecute.Start:
		// Add first motion/command steps for the production cycle.
		;
		
	E_EM_Lift_Seq_ProductionExecute.Ready:
		// Sequence complete; state complete is set automatically to omac.
		;
	E_EM_Lift_Seq_ProductionExecute.Error:
		;
END_CASE

// Return sequencer status to PackML state handler.
_m_ProductionExecute := s_fbSeqControl.m_getResult(TO_STRING(s_eSeq));
END_METHOD

METHOD _m_ProductionStarting : ITF_FB_SeqControl
VAR_INPUT
	i_bCmdRestart : BOOL;
END_VAR
VAR_INST
	s_fbSeqControl  : FB_SeqControl;
	s_eSeq 			: E_EM_Lift_Seq_ProductionStarting;
	s_stHomingOptions : ST_HomingOptions;
END_VAR

// Sequencer bookkeeping (current step and entry handling).
s_fbSeqControl(
	i_bReqStart:= i_bCmdRestart, 
	i_rnActSeqStep:= s_eSeq, 
	i_sActSeqStep:= TO_STRING(s_eSeq));
	
// Production start sequence: home, enable, and move to a known start position.
CASE s_eSeq OF 
	E_EM_Lift_Seq_ProductionStarting.Idle:
		// Wait for start command from PackML.
		;
	E_EM_Lift_Seq_ProductionStarting.Start:
		// Current logic: if axis reports homed, re-run reference; otherwise enable.
		// Adjust this decision to match your homing policy.
		IF s_cmMotorLift.p_bStaHomed THEN
			s_fbSeqControl.m_ReqStep(E_EM_Lift_Seq_ProductionStarting.ReferenceDrive);
		ELSE	
			s_fbSeqControl.m_ReqStep(E_EM_Lift_Seq_ProductionStarting.EnableDrive);
		END_IF
	
	E_EM_Lift_Seq_ProductionStarting.ReferenceDrive:
		// Configure homing behavior for this axis.
		s_stHomingOptions.ClearPositionLag := TRUE;
		s_stHomingOptions.SearchDirection := MC_Direction.MC_Positive_Direction;
		s_stHomingOptions.SearchVelocity := 500;
		s_stHomingOptions.SyncDirection := MC_Direction.MC_Negative_Direction;
		s_stHomingOptions.SyncVelocity := 100;
		s_stHomingOptions.ReferenceMode := E_EncoderReferenceMode.ENCODERREFERENCEMODE_DEFAULT;
		
		// Start homing on entry and wait until it completes.
		IF s_cmMotorLift.m_Home(
			i_bCmdExecute:= s_fbSeqControl.p_bStaEntry, 
			i_bForceReference:= TRUE, 
			i_eHomingMode:= MC_HomingMode.MC_Direct, 
			i_eBufferMode:= MC_BufferMode.MC_Aborting, 
			i_fPosition:= 0.0, 
			i_stOptions:= s_stHomingOptions, 
			i_sLogHint:= 'Starting')
		THEN
			s_fbSeqControl.m_ReqStep(E_EM_Lift_Seq_ProductionStarting.EnableDrive);
		END_IF
	E_EM_Lift_Seq_ProductionStarting.EnableDrive:
		// Power on the drive before any absolute move commands.
		IF s_cmMotorLift.m_PowerOn() THEN
			s_fbSeqControl.m_ReqStep(E_EM_Lift_Seq_ProductionStarting.MoveToStartPos);
		END_IF
		
	E_EM_Lift_Seq_ProductionStarting.MoveToStartPos:
		// Move to a defined start position for production.
		IF s_cmMotorLift.m_MoveAbsolute(
								i_bCmdExecute:= s_fbSeqControl.p_bStaEntry, 
								i_fAcceleration:= 500, 
								i_fDeceleration:= 500, 
								i_fJerk:= 5000, 
								i_fSpeed:= 100, 
								i_fPosition:= 100, 
								i_eBufferMode:= MC_BufferMode.MC_Aborting, 
								i_sLogHint:= 'Starting, move to startposition')	
		THEN
			s_fbSeqControl.m_ReqStep(E_EM_Lift_Seq_ProductionStarting.Ready);
		END_IF
		
	E_EM_Lift_Seq_ProductionStarting.Ready:
		// Start sequence complete; ready for Execute state.
		;
	E_EM_Lift_Seq_ProductionStarting.Error:
		;
END_CASE

// Return sequencer status to PackML state handler.
_m_ProductionStarting := s_fbSeqControl.m_getResult(TO_STRING(s_eSeq));
END_METHOD

METHOD _m_SeqStopServos : ITF_FB_SeqControl
VAR_INPUT
	i_bCmdRestart : BOOL;
END_VAR
VAR_INST
	s_fbSeqControl  : FB_SeqControl;
	s_eSeq 			: E_EM_Lift_Seq_StopServos;
END_VAR
// Sequencer bookkeeping (current step and entry handling).
s_fbSeqControl(
	i_bReqStart:= i_bCmdRestart, 
	i_rnActSeqStep:= s_eSeq, 
	i_sActSeqStep:= TO_STRING(s_eSeq));


// Stop sequence - bring the servo to a safe, powered-off state.
CASE s_eSeq OF
	E_EM_Lift_Seq_StopServos.Idle:
		// Wait for stop request from PackML or safety logic.
		;
		
	E_EM_Lift_Seq_StopServos.Start:
		// Issue emergency stop to decelerate as fast as possible.
		IF s_cmMotorLift.m_EmrStop(i_bCmdExecute := s_fbSeqControl.p_bStaEntry) THEN
			s_fbSeqControl.m_ReqStep(E_EM_Lift_Seq_StopServos.PowerOffServo);
		ELSIF s_fbSeqControl.p_tmStepTime > T#200MS THEN	
			// Not stopped in expected time; continue with power-off.
			s_fbSeqControl.m_ReqStep(E_EM_Lift_Seq_StopServos.PowerOffServo);
		END_IF
		
	E_EM_Lift_Seq_StopServos.PowerOffServo :	
		// Remove drive power after the stop request.
		IF s_cmMotorLift.m_PowerOff() THEN
			s_fbSeqControl.m_ReqStep(E_EM_Lift_Seq_StopServos.Ready);
		ELSIF s_fbSeqControl.p_tmStepTime > T#200MS THEN
			// Not powered off in expected time; end sequence anyway.
			s_fbSeqControl.m_ReqStep(E_EM_Lift_Seq_StopServos.Ready);
		END_IF
			
		
	E_EM_Lift_Seq_StopServos.Ready:
		// Stop sequence complete.
		;
	E_EM_Lift_Seq_StopServos.Error:
		;
END_CASE

// Return sequencer status to PackML state handler.
_m_SeqStopServos := s_fbSeqControl.m_getResult(TO_STRING(s_eSeq));
END_METHOD

METHOD PROTECTED _m_Starting : BOOL // Return state complete when state is ready
VAR_INPUT
	i_bCmdRestart	: BOOL;	//First cycle of this state
	i_eActMode 		: E_PackML_Mode;
END_VAR
VAR_INST
	s_fbSeqControl 	: FB_SeqControl;
	s_eSeq			: E_EM_InfeedConveyor_Seq_ProductionStarting;
END_VAR
// PackML Starting: run production-start sequencer in Production mode.
IF i_eActMode = E_PackML_Mode.Production THEN
	_m_Starting := _m_ProductionStarting(i_bCmdRestart := i_bCmdRestart).p_bStaReady;
ELSE
	_m_Starting := TRUE;
END_IF
END_METHOD

METHOD PROTECTED _m_Stopping : BOOL // Return state complete when state is ready
VAR_INPUT
	i_bCmdRestart	: BOOL;	//First cycle of this state
	i_eActMode 		: E_PackML_Mode;
END_VAR
// Abort and disable servo
// PackML Stopping reuses the stop-sequence to safely disable the servo.
_m_Stopping	:= _m_SeqStopServos(i_bCmdRestart := i_bCmdRestart).p_bStaReady;
END_METHOD

END_FUNCTION_BLOCK

// ---- POUs/1_Management_Layer/FB_HMI_AlarmCollector.TcPOU
FUNCTION_BLOCK FB_HMI_AlarmCollector EXTENDS FB_Base
VAR_INPUT
	i_itfAlarmCollector		: ITF_AlarmCollector; // Alarm collector interface (source of active alarms).
END_VAR
VAR_OUTPUT
END_VAR
VAR

	s_stHmi					: ST_HmiAlarmList; // HMI alarm list output structure.

	s_aitfActiveAlarms		: ARRAY[1..Param_Alarms.c_nMaxNrOfListEntries] OF ITF_AlarmHandler; // Active alarm interfaces.
	s_nIndex				: UINT; // Loop index for list building.
END_VAR

// Call base
SUPER^();

METHOD PROTECTED _m_Hmi
VAR_INST
	s_itfHighestActiveAlarm : ITF_AlarmHandler;
END_VAR
// Build HMI alarm list and highest active alarm from the collector.
IF i_itfAlarmCollector = 0 THEN
	// No collector attached: clear outputs and exit.
	s_itfHighestActiveAlarm := 0;
	s_stHmi.sHighestActiveAlarm := '';
	FOR s_nIndex := 1 TO Param_Alarms.c_nMaxNrOfListEntries DO
		s_stHmi.asAlarmList[s_nIndex] := '';
	END_FOR
	RETURN;
END_IF

// Reset outputs before (re)building the list
s_itfHighestActiveAlarm := 0;
s_stHmi.sHighestActiveAlarm := '';
FOR s_nIndex := 1 TO Param_Alarms.c_nMaxNrOfListEntries DO
	s_stHmi.asAlarmList[s_nIndex] := '';
END_FOR

// Fetch active alarms from collector into local array.
i_itfAlarmCollector.m_GetActiveAlarms(q_aitfAlarms => s_aitfActiveAlarms);

FOR s_nIndex := 1 TO Param_Alarms.c_nMaxNrOfListEntries DO
	IF s_aitfActiveAlarms[s_nIndex] <> 0 AND_THEN s_aitfActiveAlarms[s_nIndex].p_bStaRaised THEN
		// Track highest severity alarm for quick HMI display.
		IF (s_itfHighestActiveAlarm = 0) THEN
			s_itfHighestActiveAlarm := s_aitfActiveAlarms[s_nIndex];
			s_stHmi.sHighestActiveAlarm := s_aitfActiveAlarms[s_nIndex].p_sEventText;
		ELSIF s_itfHighestActiveAlarm <> 0 AND_THEN (s_aitfActiveAlarms[s_nIndex].p_eAlarmState > s_itfHighestActiveAlarm.p_eAlarmState) THEN
			s_itfHighestActiveAlarm := s_aitfActiveAlarms[s_nIndex];
			s_stHmi.sHighestActiveAlarm := s_aitfActiveAlarms[s_nIndex].p_sEventText;
		END_IF

		// Copy alarm text into the list for the HMI.
		s_stHmi.asAlarmList[s_nIndex] := s_aitfActiveAlarms[s_nIndex].p_sEventText;
	END_IF
END_FOR
END_METHOD

(* Main method of the FB *)
METHOD m_Main
// Main cycle: call base then update HMI alarm data.
SUPER^.m_Main();

_m_Hmi(); // Build alarm list for HMI display.
END_METHOD

END_FUNCTION_BLOCK

// ---- POUs/6_TwinCatChecks/CheckBounds.TcPOU
// Checkbounds is used to check for range overflows in the project.
// Implicitly generated code : DO NOT EDIT
FUNCTION CheckBounds : DINT
VAR_INPUT
	index, lower, upper: DINT;
END_VAR

// Implicitly generated code : Only an Implementation suggestion
{noflow}
IF  index < lower THEN
	CheckBounds := lower;
	GVL_TwinCatChecks.CheckBounds_DINT_TooLow := GVL_TwinCatChecks.CheckBounds_DINT_TooLow + 1;
	
ELSIF  index > upper THEN
	CheckBounds := upper;
	GVL_TwinCatChecks.CheckBounds_DINT_TooHigh := GVL_TwinCatChecks.CheckBounds_DINT_TooHigh + 1;
	
ELSE  
	CheckBounds := index;
END_IF
{flow}

END_FUNCTION

// ---- POUs/6_TwinCatChecks/CheckDivDInt.TcPOU
// This Function is used to avoid division by 0.
// If you integrate these functions in the PLC project, they are called before each division that occurs in the code.
// Implicitly generated code : DO NOT EDIT
FUNCTION CheckDivDInt : DINT
VAR_INPUT
	divisor:DINT;
END_VAR

// Implicitly generated code : Only an Implementation suggestion
{noflow}
IF divisor = 0 THEN
	CheckDivDInt:=1;
	GVL_TwinCatChecks.CheckDiv_DINT_DivBy0 := GVL_TwinCatChecks.CheckDiv_DINT_DivBy0 + 1;
ELSE
	CheckDivDInt:=divisor;
END_IF;
{flow}

END_FUNCTION

// ---- POUs/6_TwinCatChecks/CheckDivLInt.TcPOU
// This Function is used to avoid division by 0.
// If you integrate these functions in the PLC project, they are called before each division that occurs in the code.
// Implicitly generated code : DO NOT EDIT
FUNCTION CheckDivLInt : LINT
VAR_INPUT
	divisor:LINT;
END_VAR

// Implicitly generated code : Only an Implementation suggestion
{noflow}
IF divisor = 0 THEN
	CheckDivLInt:=1;
	GVL_TwinCatChecks.CheckDiv_LINT_DivBy0 := GVL_TwinCatChecks.CheckDiv_LINT_DivBy0 + 1;
ELSE
	CheckDivLInt:=divisor;
END_IF;
{flow}

END_FUNCTION

// ---- POUs/6_TwinCatChecks/CheckDivLReal.TcPOU
// This Function is used to avoid division by 0.
// If you integrate these functions in the PLC project, they are called before each division that occurs in the code.
// Implicitly generated code : DO NOT EDIT
FUNCTION CheckDivLReal : LREAL
VAR_INPUT
	divisor:LREAL;
END_VAR

// Implicitly generated code : Only an Implementation suggestion
{noflow}
IF divisor = 0 THEN
	CheckDivLReal:=1;
	GVL_TwinCatChecks.CheckDiv_LREAL_DivBy0 := GVL_TwinCatChecks.CheckDiv_LREAL_DivBy0 + 1;
ELSE
	CheckDivLReal:=divisor;
END_IF;
{flow}

END_FUNCTION

// ---- POUs/6_TwinCatChecks/CheckDivReal.TcPOU
// This Function is used to avoid division by 0.
// If you integrate these functions in the PLC project, they are called before each division that occurs in the code.
// Implicitly generated code : DO NOT EDIT
FUNCTION CheckDivReal : REAL
VAR_INPUT
	divisor:REAL;
END_VAR

// Implicitly generated code : Only an Implementation suggestion
{noflow}
IF divisor = 0 THEN
	CheckDivReal:=1;
	GVL_TwinCatChecks.CheckDiv_REAL_DivBy0 := GVL_TwinCatChecks.CheckDiv_REAL_DivBy0 + 1;
ELSE
	CheckDivReal:=divisor;
END_IF;
{flow}

END_FUNCTION

// ---- POUs/6_TwinCatChecks/CheckLRangeSigned.TcPOU
// CheckLRangeSigned checks subrange types of the type LINT.
// The purpose of this monitoring function is to deal with range bound violations as appropriate.
// Implicitly generated code : DO NOT EDIT
FUNCTION CheckLRangeSigned : LINT
VAR_INPUT
	value, lower, upper: LINT;
END_VAR

// Implicitly generated code : Only an Implementation suggestion
{noflow}
IF (value < lower) THEN
	CheckLRangeSigned := lower;
	GVL_TwinCatChecks.CheckRange_LINT_TooLow := GVL_TwinCatChecks.CheckRange_LINT_TooLow + 1;
ELSIF(value > upper) THEN
	CheckLRangeSigned := upper;
	GVL_TwinCatChecks.CheckRange_LINT_TooHigh := GVL_TwinCatChecks.CheckRange_LINT_TooHigh + 1;
ELSE
	CheckLRangeSigned := value;
END_IF
{flow}

END_FUNCTION

// ---- POUs/6_TwinCatChecks/CheckLRangeUnsigned.TcPOU
// CheckLRangeUnsigned checks subrange types of the type LWORD, ULINT.
// The purpose of this monitoring function is to deal with range bound violations as appropriate.
// Implicitly generated code : DO NOT EDIT
FUNCTION CheckLRangeUnsigned : ULINT
VAR_INPUT
	value, lower, upper: ULINT;
END_VAR

// Implicitly generated code : Only an Implementation suggestion
{noflow}
IF (value < lower) THEN
	CheckLRangeUnsigned := lower;
	GVL_TwinCatChecks.CheckRange_ULINT_TooLow := GVL_TwinCatChecks.CheckRange_ULINT_TooLow + 1;
ELSIF(value > upper) THEN
	CheckLRangeUnsigned := upper;
	GVL_TwinCatChecks.CheckRange_ULINT_TooHigh := GVL_TwinCatChecks.CheckRange_ULINT_TooHigh + 1;
ELSE
	CheckLRangeUnsigned := value;
END_IF
{flow}

END_FUNCTION

// ---- POUs/6_TwinCatChecks/CheckPointer.TcPOU
// This Function is used to monitor the memory acces of pointers during runtime.
// The purpose of the CheckPointer function is to check whether the transferred pointer points to a valid memory address, and whether the orientation of the referenced memory area matches the type of variable to which the pointer points.
// If both conditions are met, the pointer itself is returned. Otherwise, the function should perform proper error handling.
// Implicitly generated code : DO NOT EDIT
FUNCTION CheckPointer : POINTER TO BYTE
VAR_INPUT 
	ptToTest : POINTER TO BYTE; // Destination address of the pointer
	iSize : DINT;		        // Size of the type the pointer points to. (e.g: 20 for POINTER TO ARRAY [0..9] OF INT) 
	iGran : DINT;		        // Granularity of the pointer access. This is the size of the biggest non-structured data type in the type the pointer points to. (e.g: 2 for POINTER TO ARRAY [0..9] OF INT)
	bWrite: BOOL;		        // Indicates read or write Access. TRUE = write access.
END_VAR

// No standard way of implementation. Fill your own code here
{noflow}
CheckPointer := ptToTest;
{flow}

END_FUNCTION

// ---- POUs/6_TwinCatChecks/CheckRangeSigned.TcPOU
// CheckRangeSigned checks subrange types of the type SINT, INT, DINT
// The purpose of this monitoring function is to deal with range bound violations as appropriate.
// Implicitly generated code : DO NOT EDIT
FUNCTION CheckRangeSigned : DINT
VAR_INPUT
	value, lower, upper: DINT;
END_VAR

// Implicitly generated code : Only an Implementation suggestion
{noflow}
IF (value < lower) THEN
	CheckRangeSigned := lower;
	GVL_TwinCatChecks.CheckRange_DINT_TooLow := GVL_TwinCatChecks.CheckRange_DINT_TooLow + 1;
ELSIF(value > upper) THEN
	CheckRangeSigned := upper;
	GVL_TwinCatChecks.CheckRange_DINT_TooHigh := GVL_TwinCatChecks.CheckRange_DINT_TooHigh + 1;
ELSE
	CheckRangeSigned := value;
END_IF
{flow}

END_FUNCTION

// ---- POUs/6_TwinCatChecks/CheckRangeUnsigned.TcPOU
// CheckRangeUnsigned checks subrange types of the type BYTE, WORD, DWORD, USINT, UINT, UDINT.
// The purpose of this monitoring function is to deal with range bound violations as appropriate.
// Implicitly generated code : DO NOT EDIT
FUNCTION CheckRangeUnsigned : UDINT
VAR_INPUT
	value, lower, upper: UDINT;
END_VAR

// Implicitly generated code : Only an Implementation suggestion
{noflow}
IF (value < lower) THEN
	CheckRangeUnsigned := lower;
	GVL_TwinCatChecks.CheckRange_UDINT_TooLow := GVL_TwinCatChecks.CheckRange_UDINT_TooLow + 1;
ELSIF(value > upper) THEN
	CheckRangeUnsigned := upper;
	GVL_TwinCatChecks.CheckRange_UDINT_TooHigh := GVL_TwinCatChecks.CheckRange_UDINT_TooHigh + 1;
ELSE
	CheckRangeUnsigned := value;
END_IF
{flow}

END_FUNCTION

// ---- GlobalTextList.TcGTLO
TEXTLIST GlobalTextList
  354 = '%s'
  612 = '.bAlwStateChange'
  203 = 'ActMode'
  31 = 'ActState'
  943 = 'ActSubState'
  923 = 'Actual mode'
  256 = 'Actual mode:'
  117 = 'Actual state'
  42 = 'Actual state:'
  581 = 'Alarms'
  751 = 'AlwStateChange'
  467 = 'bAlwStateChange'
  201 = 'bModeChangeInProcess'
  267 = 'bStateComplete'
  474 = 'eActMode'
  651 = 'eActState'
  49 = 'emLogicExample Alarms List'
  985 = 'emLogicExample2 Alarms List'
  747 = 'eReqMode'
  729 = 'eReqState'
  697 = 'Hoofdmenu'
  438 = 'Infeed'
  39 = 'InstancePath'
  299 = 'InstancePath[INDEX]'
  782 = 'Mode Production'
  492 = 'nActSubState'
  652 = 'PackML'
  670 = 'PackML Instance Path'
  499 = 'ReqState'
  490 = 'Reset'
  356 = 'SC'
  705 = 'Simulation'
  864 = 'Start'
  94 = 'State'
  347 = 'State Time'
  64 = 'StateTime'
  796 = 'Stop'
  740 = 'tmStateTime'
  681 = 'unMachine100 Alarms List'
END_TEXTLIST

// ---- VISUs/HMI_Button.TcVIS
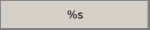
VISUALIZATION HMI_Button  // 150x30
VAR_INPUT
	i_sText : STRING;
END_VAR
VAR_IN_OUT
	iq_stButton : ST_HmiButton;
END_VAR
    Button (0,0 150x30), "%s", text variable: i_sText, pressed state: iq_stButton.stToHmi.bProcessState, invisible if: iq_stButton.stToHmi.bInvisible, input disabled if: not iq_stButton.stToHmi.bEnabled
        tap iq_stButton.stFromHmi.bPressed
END_VISUALIZATION

// ---- VISUs/Header.TcVIS
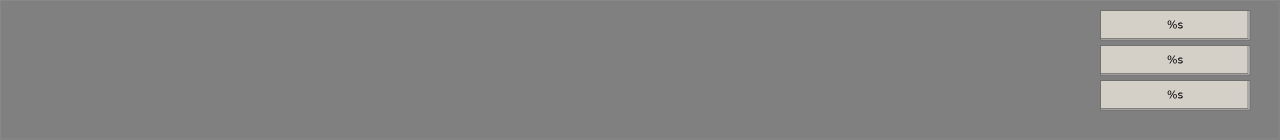
VISUALIZATION Header  // 1280x140
    Rectangle (0,0 1280x140)
    Frame (1100,10 150x30)
        shows HMI_Button(i_sText := 'Start', iq_stButton := GVL_Modules.g_fbHmiMachCtrlsManager.s_fbBtnReqStart.s_stHmi)
    Frame (1100,45 150x30)
        shows HMI_Button(i_sText := 'Stop', iq_stButton := GVL_Modules.g_fbHmiMachCtrlsManager.s_fbBtnReqStop.s_stHmi)
    Frame (1100,80 150x30)
        shows HMI_Button(i_sText := 'Reset', iq_stButton := GVL_Modules.g_fbHmiMachCtrlsManager.s_fbBtnReqReset.s_stHmi)
END_VISUALIZATION

// ---- VISUs/Page_Main.TcVIS
VISUALIZATION Page_Main  // 1080x660, background image 
END_VISUALIZATION

// ---- VISUs/Page_Alarms.TcVIS
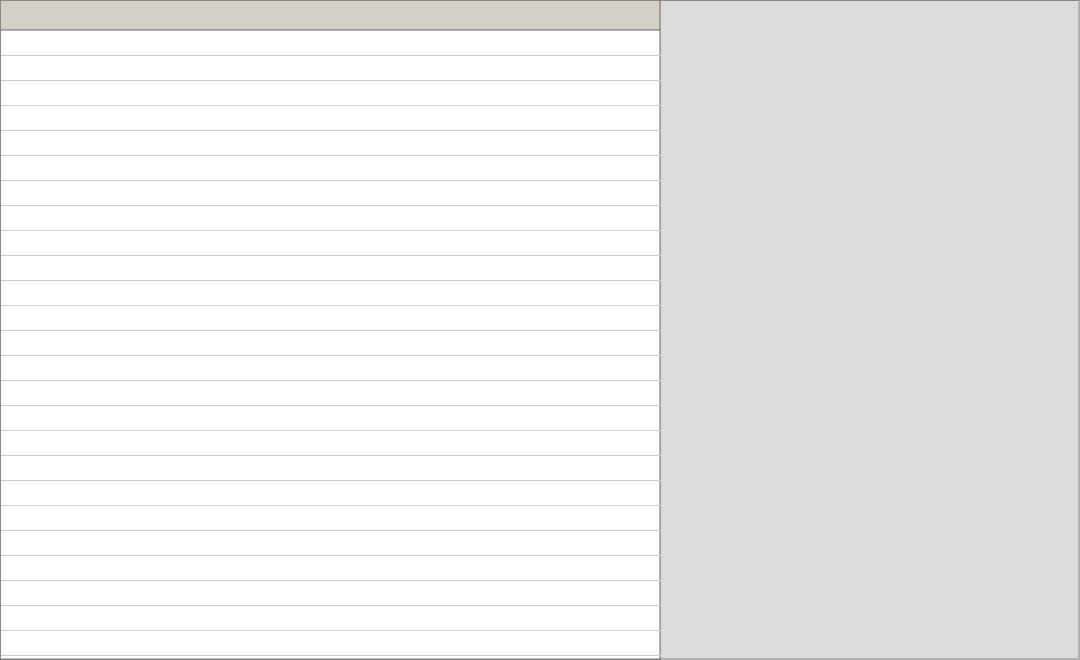
VISUALIZATION Page_Alarms  // 1080x660, background image 
    Table (0,0 660x660), data array: GVL_Modules.g_unMachine.s_stHmi.fbHmiAlarmCollector.s_stHmi.asAlarmList
        p3854506369: GVL_Modules.g_unMachine.s_stHmi.fbHmiAlarmCollector.s_stHmi.asAlarmList[INDEX]
        p1014161805: Param_Alarms.c_nMaxNrOfListEntries - 1 + INT#1
END_VISUALIZATION

// ---- VISUs/Page_Infeed.TcVIS
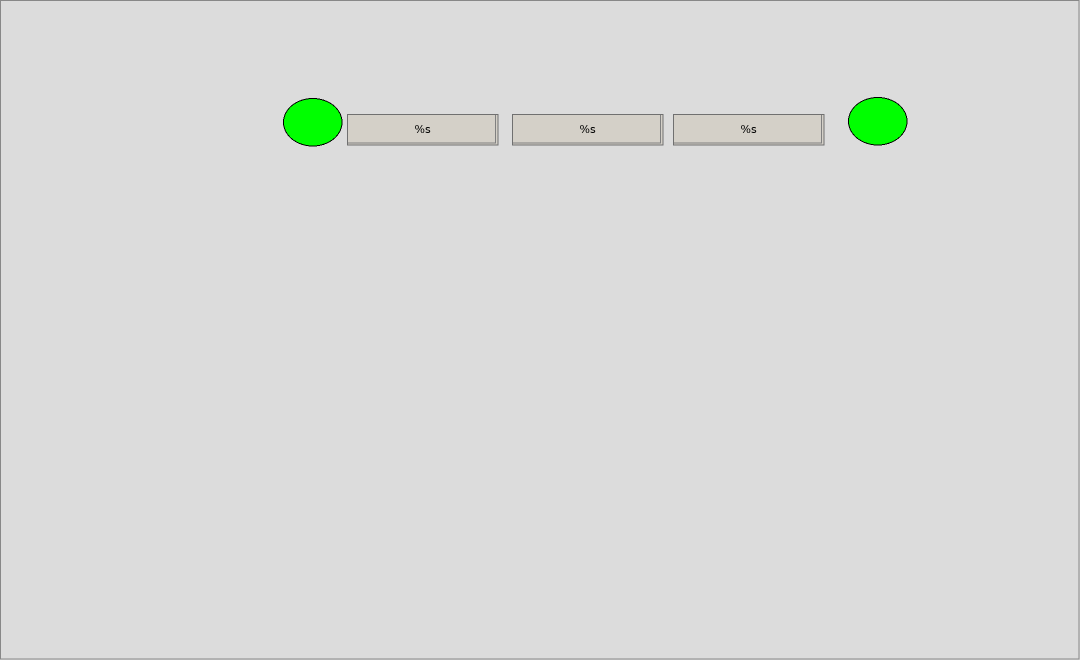
VISUALIZATION Page_Infeed  // 1080x660, background image 
    Frame (347,114 151x31)
        shows HMI_Button(i_sText := 'Open', iq_stButton := GVL_Modules.g_emInfeedConveyor.s_cmDoor.s_stHmi.btnOpenDoor.s_stHmi)
    Frame (673,114 151x31)
        shows HMI_Button(i_sText := 'Close', iq_stButton := GVL_Modules.g_emInfeedConveyor.s_cmDoor.s_stHmi.btnCloseDoor.s_stHmi)
    Frame (512,114 151x31)
        shows HMI_Button(i_sText := 'Stop', iq_stButton := GVL_Modules.g_emInfeedConveyor.s_cmDoor.s_stHmi.btnStopDoor.s_stHmi)
    Ellipse (283,98 59x48), colour toggle: not GVL_Modules.g_emInfeedConveyor.s_cmDoor.s_stHmi.bStaDoorOpen
    Ellipse (848,97 59x48), colour toggle: not GVL_Modules.g_emInfeedConveyor.s_cmDoor.s_stHmi.bStaDoorCLosed
END_VISUALIZATION

// ---- VISUs/Page_PackML.TcVIS
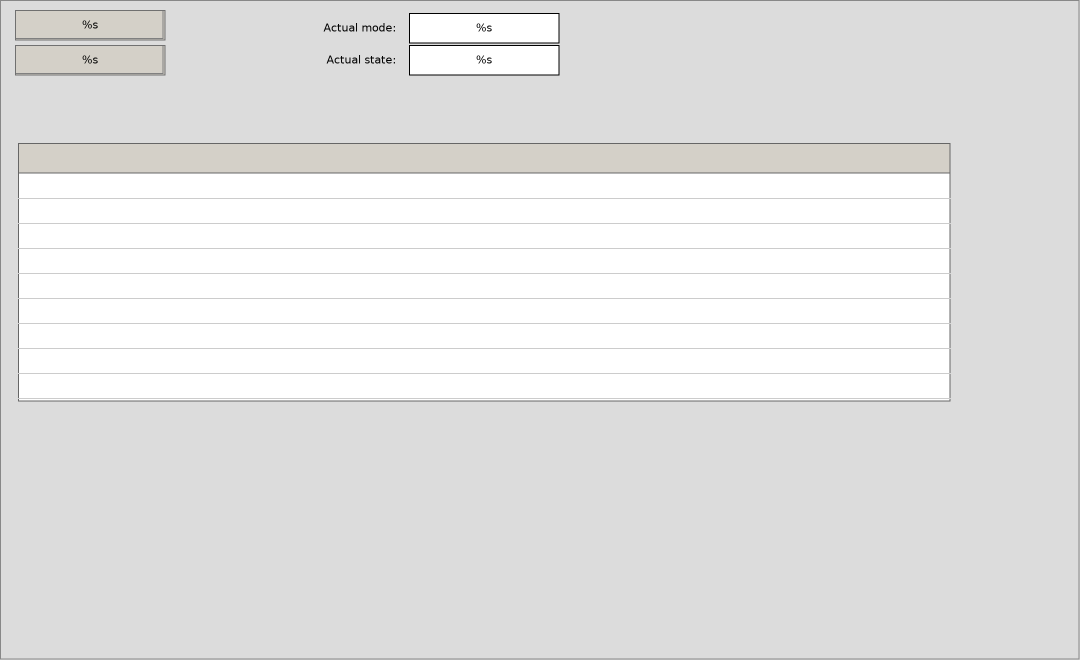
VISUALIZATION Page_PackML  // 1080x660, background image 
    Frame (15,10 150x30)
        shows HMI_Button(i_sText := 'Production', iq_stButton := GVL_Modules.g_fbHmiMachCtrlsManager.s_fbBtnReqProduction.s_stHmi)
    Frame (15,45 150x30)
        shows HMI_Button(i_sText := 'Manual', iq_stButton := GVL_Modules.g_fbHmiMachCtrlsManager.s_fbBtnReqManual.s_stHmi)
    Rectangle (249,13 150x30), "Actual mode:"
    Rectangle (249,45 150x30), "Actual state:"
    Rectangle (409,45 150x30), "%s", text variable: GVL_Modules.g_fbHmiMachCtrlsManager.s_eActState
    Rectangle (409,13 150x30), "%s", text variable: GVL_Modules.g_fbHmiMachCtrlsManager.s_eActMode
    Table (18,143 932x258), data array: GVL_Modules.g_fbPackMLstatusManager.q_astPackML_status
        p3854506369: GVL_Modules.g_fbPackMLstatusManager.q_astPackML_status[INDEX].sPackML_InstancePath
        p1014161805: GSBF_Common.Param_packML.c_nMaxNrOfChildren - 1 + INT#1
        p1892666644: GVL_Modules.g_fbPackMLstatusManager.q_astPackML_status[INDEX].eActMode
        p338671338: GVL_Modules.g_fbPackMLstatusManager.q_astPackML_status[INDEX].eReqMode
        p2170511999: GVL_Modules.g_fbPackMLstatusManager.q_astPackML_status[INDEX].eActState
        p3723444502: GVL_Modules.g_fbPackMLstatusManager.q_astPackML_status[INDEX].eReqState
        p1218418051: GVL_Modules.g_fbPackMLstatusManager.q_astPackML_status[INDEX].bStateComplete
        p746581629: GVL_Modules.g_fbPackMLstatusManager.q_astPackML_status[INDEX].nActSubState
        p3104783080: GVL_Modules.g_fbPackMLstatusManager.q_astPackML_status[INDEX].bAlwStateChange
        p2501879983: GVL_Modules.g_fbPackMLstatusManager.q_astPackML_status[INDEX].bModeChangeInProcess
        p7306298: GVL_Modules.g_fbPackMLstatusManager.q_astPackML_status[INDEX].stReqCntrlCmd
        p1933151965: GVL_Modules.g_fbPackMLstatusManager.q_astPackML_status[INDEX].eActCntrlCmd
        p3863566920: GVL_Modules.g_fbPackMLstatusManager.q_astPackML_status[INDEX].bStateEntry
        p2192122294: GVL_Modules.g_fbPackMLstatusManager.q_astPackML_status[INDEX].bStateChangeInProcess
        p400160035: GVL_Modules.g_fbPackMLstatusManager.q_astPackML_status[INDEX].tmStateTime
        p1265227338: GVL_Modules.g_fbPackMLstatusManager.q_astPackML_status[INDEX].nReqSubState
        p3726181087: GVL_Modules.g_fbPackMLstatusManager.q_astPackML_status[INDEX].bSubStateEntry
        p3136911649: GVL_Modules.g_fbPackMLstatusManager.q_astPackML_status[INDEX].bChildrenStateComplete
        p290089404: State Time
END_VISUALIZATION

// ---- VISUs/Visualization.TcVIS
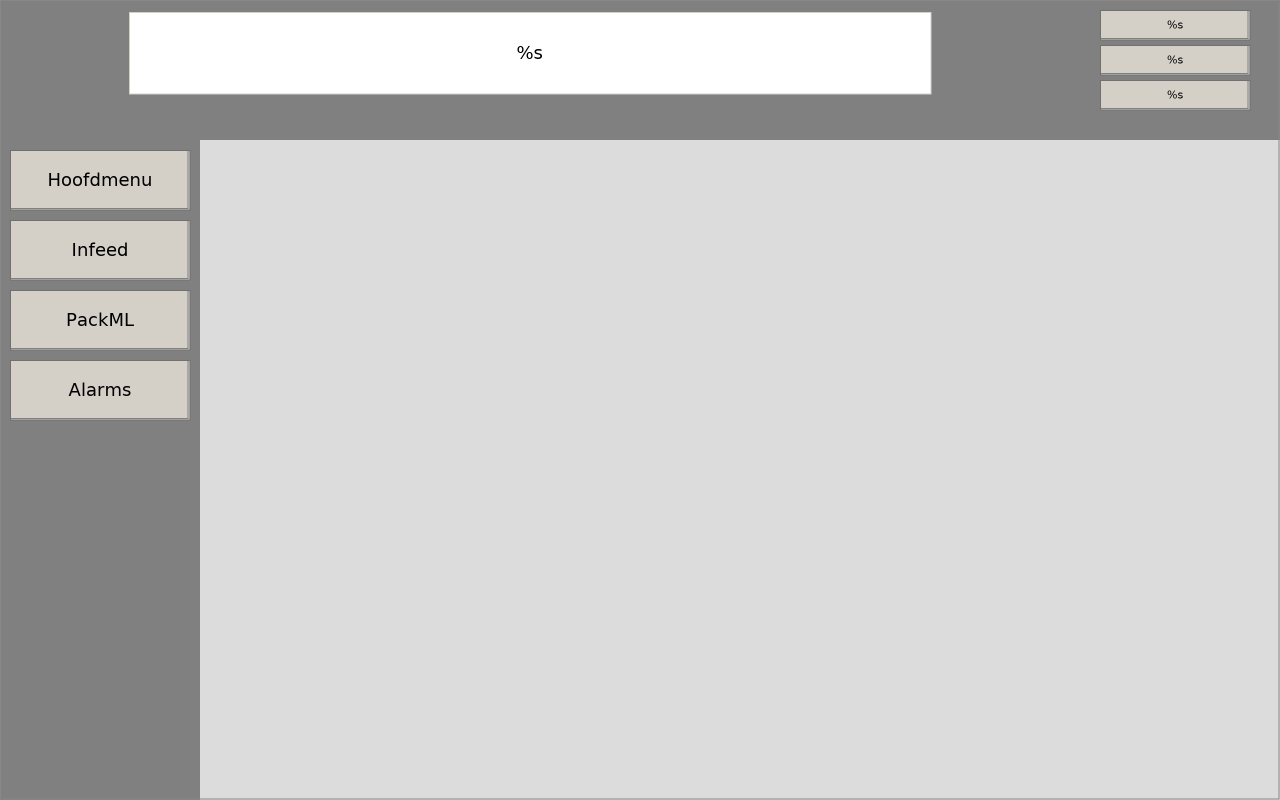
VISUALIZATION Visualization  // 1280x800
VAR_IN_OUT
END_VAR
VAR
	s_nPageIndex : DINT;
END_VAR
    Rectangle (0,140 200x660)
    Frame (0,0 1280x140)
        shows Header()
    Button (10,150 180x60), "Hoofdmenu", pressed state: s_nPageIndex = 0
        OnMouseClick: execute { s_nPageIndex := 0; }
    Button (10,220 180x60), "Infeed", pressed state: s_nPageIndex = 1
        OnMouseClick: execute { s_nPageIndex := 1; }
    Button (10,290 180x60), "PackML", pressed state: s_nPageIndex = 2
        OnMouseClick: execute { s_nPageIndex := 2; }
    Button (10,360 180x60), "Alarms", pressed state: s_nPageIndex = 3
        OnMouseClick: execute { s_nPageIndex := 3; }
    Frame (200,140 1080x660), frame switch variable: s_nPageIndex
        shows Page_Main()
        shows Page_Infeed()
        shows Page_PackML()
        shows Page_Alarms()
    Textfield (129,12 802x82), "%s", text variable: GVL_Modules.g_unMachine.s_stHmi.fbHmiAlarmCollector.s_stHmi.sHighestActiveAlarm, colour toggle: GVL_Modules.g_unMachine.s_fbAlarmCollector.p_bStaRaised
        OnMouseClick: execute { s_npageIndex := 3; }
END_VISUALIZATION
